TYPE ST_Params :
STRUCT
	fEncoderOffset : LREAL;
END_STRUCT
END_TYPE

(* stored: Version 1.1.0.1, ProductVersion 3.1.4024.12
   DUT ST_Params: Id {17456da7-9450-45ee-9e90-f87c5ba29ab0} *)
